FUNCTION_BLOCK Tank
VAR_INPUT
	diMixer_Running : BOOL;
	diMixer_Error : BOOL;
END_VAR
VAR_OUTPUT
	doMixer_Start : BOOL;
END_VAR
VAR_IN_OUT
	ioTank : TTank;
END_VAR
VAR

END_VAR

Engine(iRunning:=diMixer_Running, iError:=diMixer_Error, Engine:=ioTank.Mixer);
Engine.oRun:=doMixer_Start

END_FUNCTION_BLOCK

(* stored: Version 1.1.0.1, ProductVersion 3.1.4024.12
   POU Tank: Id {f84ad52f-e512-422e-be18-b265eb0ae589}, SpecialFunc None *)
